FUNCTION_BLOCK AxisControl
VAR
	
	// Axis Reference
	_Axis					: ARRAY [1.._NumberOfAxes] OF AXIS_REF;		
	
	// Internal Variables
	_i						: UINT := 0;
	_InputToggle			: BOOL := FALSE;
	_LocalState				: UINT := 0;
	_InternalCounter		: UDINT := 0;
	_InternalCounterMax		: UDINT := 1000;
	_ErrorIDPrevious		: ARRAY [1.._NumberOfAxes] OF UDINT;
	_ErrorCount				: ARRAY [1.._NumberOfAxes] OF UINT;
	_BusyMoving				: ARRAY [1.._NumberOfAxes] OF BOOL;
	_BusyStopping			: ARRAY [1.._NumberOfAxes] OF BOOL;
	_CommandDone			: BOOL := FALSE;
	_CurrentPosition		: ARRAY [1.._NumberOfAxes] OF LREAL;
	_CurrentPositionModulo	: ARRAY [1.._NumberOfAxes] OF LREAL;
	
	// Internal Functions
	_ErrorCountTrigger		: R_TRIG;
	_DelayTimer				: TON;	
	
	// Axis States (STRUCTURE Declaration)
	_Status					: ARRAY [1.._NumberOfAxes] OF AxisStatus;
	
	// Motion Functions Blocks
	_Enable					: ARRAY [1.._NumberOfAxes] OF MC_Power;
	_Reset					: ARRAY [1.._NumberOfAxes] OF MC_Reset;
	_ReadStatus				: ARRAY [1.._NumberOfAxes] OF MC_ReadStatus;
	_WriteParameter			: MC_WriteParameter;	
	_MoveAbs1				: MC_MoveAbsolute;
	_MoveAbs2				: MC_MoveAbsolute;
	_MoveRel1				: MC_MoveRelative;
	_MoveRel2				: MC_MoveRelative;
	_MoveVel1				: MC_MoveVelocity;
	_MoveVel2				: MC_MoveVelocity;
	_StopWeak				: MC_Halt;
	_StopStrong				: MC_Stop;
		
END_VAR
VAR CONSTANT
	
	_NumberOfAxes			: UINT := 3;

END_VAR

METHOD AutoErrorCheckAndReset : BOOL
VAR_INPUT
	AxisID			: UINT;	
END_VAR

// Automatically check for errors on the NC axis, then reset them
// Use with caution, this could cause damage to a physical system if implemented without care

_ReadStatus[AxisID](Axis := _Axis[AxisID]);
_Reset[AxisID](Axis := _Axis[AxisID]);
_ErrorCountTrigger(CLK := _Status[AxisID]._Error);

IF _ErrorCountTrigger.Q THEN
	_ErrorCount[AxisID] := _ErrorCount[AxisID] + 1;
END_IF

IF _Status[AxisID]._Error THEN
	_LocalState := 0;
	_Reset[AxisID].Execute := TRUE;
	IF _Reset[AxisID].Done THEN
		_Reset[AxisID].Execute := FALSE;
		AutoErrorCheckAndReset := TRUE;
	END_IF
END_IF
END_METHOD

PROPERTY AxisStatus : ARRAY [1.._NumberOfAxes] OF AxisStatus
GET
AxisStatus := _Status;
END_GET
SET
END_SET
END_PROPERTY

METHOD CheckForErrors : BOOL
VAR_INPUT	
	AxisID			: UINT;
END_VAR

// Check for errors on the NC axis

_ReadStatus[AxisID](Axis := _Axis[AxisID]);
_ErrorCountTrigger(CLK := _Status[AxisID]._Error);

IF _ErrorCountTrigger.Q THEN
	_ErrorCount[AxisID] := _ErrorCount[AxisID] + 1;
END_IF

IF _Status[AxisID]._Error THEN
	_LocalState := 0;
	CheckForErrors := TRUE;
END_IF
END_METHOD

PROPERTY CurrentPosition : ARRAY [1.._NumberOfAxes] OF LREAL
GET
CurrentPosition := _CurrentPosition;
END_GET
SET
END_SET
END_PROPERTY

PROPERTY CurrentPositionModulo : ARRAY [1.._NumberOfAxes] OF LREAL
GET
CurrentPositionModulo := _CurrentPositionModulo;
END_GET
SET
END_SET
END_PROPERTY

METHOD CyclicUpdate : BOOL
VAR_INPUT
END_VAR

// Update method needs to be called cyclically

_InputToggle := NOT(_InputToggle);

FOR _i := 1 TO _NumberOfAxes DO
	
	_Enable[_i]		(Axis := _Axis[_i]);
	_Reset[_i]		(Axis := _Axis[_i]);
	
	_ReadStatus[_i]
	(
		Axis 					:= _Axis[_i],
		Enable 					:= TRUE,
		Error 					=> _Status[_i]._Error,
		ErrorID 				=> _Status[_i]._ErrorID,
		ErrorStop 				=> _Status[_i]._ErrorStop,
		Disabled 				=> _Status[_i]._Disabled,
		Stopping 				=> _Status[_i]._Stopping,
		StandStill 				=> _Status[_i]._StandStill,
		DiscreteMotion 			=> _Status[_i]._DiscreteMotion,
		ContinuousMotion 		=> _Status[_i]._ContinuousMotion,
		SynchronizedMotion	 	=> _Status[_i]._SynchronizedMotion,
		Homing 					=> _Status[_i]._Homing,
		ConstantVelocity		=> _Status[_i]._ConstantVelocity,
		Accelerating 			=> _Status[_i]._Accelerating,
		Decelerating 			=> _Status[_i]._Decelerating,
		Status 					=> _Status[_i]._Status
	);
	
	_BusyMoving[_i] :=
	(
		_ReadStatus[_i].DiscreteMotion OR
		_ReadStatus[_i].ConstantVelocity OR
		_ReadStatus[_i].SynchronizedMotion
	);
	
	_BusyStopping[_i] :=
	(
		_ReadStatus[_i].Stopping
	);
	
	IF _Status[_i]._ErrorID <> 0 THEN
		_ErrorIDPrevious[_i] := _Status[_i]._ErrorID;
	END_IF
			
	_CurrentPosition[_i] := _Axis[_i].NcToPlc.ActPos;
	_CurrentPositionModulo[_i] := _Axis[_i].NcToPlc.ModuloActPos;
	
END_FOR

CyclicUpdate := TRUE;
END_METHOD

PROPERTY ErrorCount : ARRAY [1.._NumberOfAxes] OF UINT
GET
ErrorCount := _ErrorCount;
END_GET
SET
END_SET
END_PROPERTY

METHOD Halt : BOOL
VAR_INPUT
	AxisID			: UINT;
END_VAR

// Halts the axis, NOT locking the axis from further commands during its process

_StopWeak(Axis := _Axis[AxisID]);

_StopWeak.Execute			:= TRUE;

IF _StopWeak.Done THEN
	_StopWeak.Execute := FALSE;
	Halt := TRUE;
END_IF

IF _StopWeak.Error THEN
	_StopWeak.Execute := FALSE;
END_IF
END_METHOD

METHOD MoveAtVelocity : BOOL
VAR_INPUT
	AxisID			: UINT;
	Velocity		: LREAL;
	Direction		: MC_Direction;
END_VAR

// Move at a given speed in a defined direction until a stop command is activated

_MoveVel1(Axis := _Axis[AxisID]);

_MoveVel1.Velocity 			:= Velocity;
_MoveVel1.Direction			:= Direction;
_MoveVel1.Execute			:= TRUE;

IF _BusyMoving[AxisID] THEN
	_MoveVel1.Execute := FALSE;
	MoveAtVelocity := TRUE;
END_IF

IF _MoveVel1.Error THEN
	_MoveVel1.Execute := FALSE;
	MoveAtVelocity := FALSE;
END_IF
END_METHOD

METHOD MoveToPosition : BOOL
VAR_INPUT
	AxisID			: UINT;
	Position		: LREAL;
	Velocity		: LREAL;
END_VAR

// Move to a specific location at a given speed

_MoveAbs1(Axis := _Axis[AxisID]);

_MoveAbs1.Position			:= Position;
_MoveAbs1.Velocity 			:= Velocity;
_MoveAbs1.Execute			:= TRUE;

IF _MoveAbs1.Done THEN
	_MoveAbs1.Execute := FALSE;
	MoveToPosition := TRUE;
END_IF

IF _MoveAbs1.Error THEN
	_MoveAbs1.Execute := FALSE;
END_IF
END_METHOD

METHOD PowerOff : BOOL
VAR_INPUT
	Override	 	: LREAL;
	AxisID			: UINT;
END_VAR

// Disable the axis

IF Override < 0 THEN
	Override := 0;
ELSIF Override > 100 THEN
	Override := 100;	
END_IF

IF AxisID < 1 THEN
	AxisID := 1;
ELSIF AxisID > _NumberOfAxes THEN
	AxisID := 1;	
END_IF

_Enable[AxisID](Axis := _Axis[AxisID]);

_Enable[AxisID].Enable 				:= FALSE;
_Enable[AxisID].Enable_Negative 	:= FALSE;
_Enable[AxisID].Enable_Positive 	:= FALSE;
_Enable[AxisID].Override 			:= 0;

IF NOT(_Enable[AxisID].Status) THEN
	PowerOff := TRUE;
ELSIF _Enable[AxisID].Error THEN
	PowerOff := FALSE;
	_Enable[AxisID].Enable := FALSE;
END_IF
END_METHOD

METHOD PowerOffAll : BOOL
VAR_INPUT
END_VAR

// Enable all axes

FOR _i := 1 TO _NumberOfAxes BY 1 DO
	_Enable[_i](Axis := _Axis[_i]);
END_FOR

CASE _LocalState OF 
	
	0:
		_LocalState := 1;
	
	1:
		FOR _i := 1 TO _NumberOfAxes BY 1 DO
			_Enable[_i](Axis := _Axis[_i]);
			_Enable[_i].Enable := FALSE;
			_Enable[_i].Enable_Negative := FALSE;
			_Enable[_i].Enable_Positive := FALSE;
			_Enable[_i].Override := 0;
		END_FOR
		_LocalState := 2;
		
	2:
		_CommandDone := TRUE;
		FOR _i := 1 TO _NumberOfAxes BY 1 DO
			IF _Enable[_i].Status THEN
				_CommandDone := FALSE;
				_InternalCounter := _InternalCounter + 1;
			END_IF
		END_FOR
		
		IF _InternalCounter >= _InternalCounterMax THEN
			_InternalCounter := 0;
			_LocalState := 0;
			PowerOffAll := FALSE;
		END_IF
		
		IF _CommandDone THEN
			_InternalCounter := 0;
			_LocalState := 3;
		END_IF
		
	3:
		_LocalState := 0;
		PowerOffAll := TRUE;

END_CASE
END_METHOD

METHOD PowerOn : BOOL
VAR_INPUT
	Override	 	: LREAL;
	AxisID			: UINT;
END_VAR

// Enable the axis

IF Override < 0 THEN
	Override := 0;
ELSIF Override > 100 THEN
	Override := 100;	
END_IF

IF AxisID < 1 THEN
	AxisID := 1;
ELSIF AxisID > _NumberOfAxes THEN
	AxisID := 1;	
END_IF

_Enable[AxisID](Axis := _Axis[AxisID]);

_Enable[AxisID].Enable 				:= TRUE;
_Enable[AxisID].Enable_Negative 	:= TRUE;
_Enable[AxisID].Enable_Positive 	:= TRUE;
_Enable[AxisID].Override 			:= 100;

IF _Enable[AxisID].Status THEN
	PowerOn := TRUE;
ELSIF _Enable[AxisID].Error THEN
	PowerOn := FALSE;
	_Enable[AxisID].Enable := FALSE;
END_IF
END_METHOD

METHOD PowerOnAll : BOOL
VAR_INPUT
	Override		: LREAL;
END_VAR

// Enable all axes

IF Override < 0 THEN
	Override := 0;
ELSIF Override > 100 THEN
	Override := 100;	
END_IF

FOR _i := 1 TO _NumberOfAxes BY 1 DO
	_Enable[_i](Axis := _Axis[_i]);
END_FOR

CASE _LocalState OF 
	
	0:
		_LocalState := 1;
	
	1:
		FOR _i := 1 TO _NumberOfAxes BY 1 DO
			_Enable[_i](Axis := _Axis[_i]);
			_Enable[_i].Enable := TRUE;
			_Enable[_i].Enable_Negative := TRUE;
			_Enable[_i].Enable_Positive := TRUE;
			_Enable[_i].Override := Override;
		END_FOR
		_LocalState := 2;
		
	2:
		_CommandDone := TRUE;
		FOR _i := 1 TO _NumberOfAxes BY 1 DO
			IF NOT(_Enable[_i].Status) THEN
				_CommandDone := FALSE;
				_InternalCounter := _InternalCounter + 1;
			END_IF
		END_FOR
		
		IF _InternalCounter >= _InternalCounterMax THEN
			_InternalCounter := 0;
			_LocalState := 0;
			PowerOnAll := FALSE;
		END_IF
		
		IF _CommandDone THEN
			_InternalCounter := 0;
			_LocalState := 3;
		END_IF
		
	3:
		_LocalState := 0;
		PowerOnAll := TRUE;

END_CASE
END_METHOD

METHOD Reset : BOOL
VAR_INPUT
	AxisID			: UINT;
END_VAR

// Reset errors on the NC axis

IF AxisID < 1 THEN
	AxisID := 1;
ELSIF AxisID > _NumberOfAxes THEN
	AxisID := 1;	
END_IF

_Reset[AxisID](Axis := _Axis[AxisID]);

_Reset[AxisID].Execute 			:= TRUE;

IF _Reset[AxisID].Done THEN
	_Reset[AxisID].Execute := FALSE;
	Reset := TRUE;
END_IF
END_METHOD

METHOD ReversingSequence : BOOL
VAR_INPUT
	AxisID			: UINT;
	Position1				: LREAL;
	Position2				: LREAL;
	Velocity				: LREAL;
	DelayBetweenMoves		: TIME;
END_VAR

// Move to Position1, then to Position2, at a set speed with a delay between the movements

_MoveAbs1(Axis := _Axis[AxisID]);
_MoveAbs2(Axis := _Axis[AxisID]);
_DelayTimer(PT := DelayBetweenMoves);

_MoveAbs1.Position			:= Position1;
_MoveAbs1.Velocity 			:= Velocity;

_MoveAbs2.Position			:= Position2;
_MoveAbs2.Velocity 			:= Velocity;

CASE _LocalState OF
	
	0:
		_MoveAbs1.Execute := TRUE;
		IF _MoveAbs1.Done THEN
			_MoveAbs1.Execute := FALSE;
			_LocalState := 1;			
		END_IF
		
	1:
		_DelayTimer.IN := TRUE;
		IF _DelayTimer.Q THEN
			_DelayTimer.IN := FALSE;
			_LocalState := 2;
		END_IF
		
	2:
		_MoveAbs2.Execute := TRUE;
		IF _MoveAbs2.Done THEN
			_MoveAbs2.Execute := FALSE;
			_LocalState := 3;			
		END_IF
		
	3:
		_DelayTimer.IN := TRUE;
		IF _DelayTimer.Q THEN
			_DelayTimer.IN := FALSE;
			_LocalState := 4;
		END_IF
		
	4:
		_LocalState := 0;
		ReversingSequence := TRUE;

END_CASE

IF _MoveAbs1.Error OR _MoveAbs2.Error THEN
	_MoveAbs1.Execute := FALSE;
	_MoveAbs2.Execute := FALSE;
END_IF
END_METHOD

METHOD Stop : BOOL
VAR_INPUT
	AxisID			: UINT;
END_VAR

// Halts the axis, locking the axis from further commands during its process

_StopStrong(Axis := _Axis[AxisID]);

_StopStrong.Execute			:= TRUE;

IF _StopStrong.Done THEN
	_StopStrong.Execute := FALSE;
	Stop := TRUE;
END_IF

IF _StopStrong.Error THEN
	_StopStrong.Execute := FALSE;
END_IF
END_METHOD

METHOD WriteToParameter : BOOL
VAR_INPUT
	AxisID			: UINT;	
	Parameter		: MC_AxisParameter;
	Value			: LREAL;
END_VAR

IF AxisID < 1 THEN
	AxisID := 1;
ELSIF AxisID > _NumberOfAxes THEN
	AxisID := 1;	
END_IF

_WriteParameter(Axis := _Axis[AxisID]);

_WriteParameter.ParameterNumber := Parameter;
_WriteParameter.Value := Value;
_WriteParameter.Execute := TRUE;


IF _WriteParameter.Done THEN
	WriteToParameter := TRUE;
	_WriteParameter.Execute := FALSE;
ELSIF _WriteParameter.Error THEN
	WriteToParameter := FALSE;
	_WriteParameter.Execute := FALSE;
END_IF
END_METHOD

END_FUNCTION_BLOCK

(* stored: Version 1.1.0.1, ProductVersion 3.1.4024.12
   POU AxisControl: Id {0762ff6d-63f2-4251-b923-cf396e8d588b}, SpecialFunc None
   Folder Methods: Id {84cb375e-4310-4c8e-b285-59f1b782ddd6}
   Folder All Axes: Id {e7566577-33ba-4fd4-a911-8164896a8c57}
   Folder Power and Monitoring: Id {72185a63-bd61-464d-9ba5-7925e55fb430}
   Folder Single Axis: Id {6793107f-f025-4746-9720-75111f89ad08}
   Folder Movements: Id {6fc24c7c-89c4-4f59-a059-62fbfee907d6}
   Folder Brake: Id {531eff0b-604f-4c37-ace9-2958971ea826}
   Folder Position: Id {8d7c9616-e265-4389-960e-a02f0ff11726}
   Folder Velocity: Id {bd356ce1-0682-451a-8f8f-f2d75631abf0}
   Folder Power and Monitoring: Id {dada0367-7150-48df-9b09-3250334c5191}
   Folder Properties: Id {391590a4-d10f-4e23-95ce-50d1b79d7756}
   Method AutoErrorCheckAndReset: Id {c4558794-dce0-4723-8ae5-ffe53ab7450c}
   Property AxisStatus: Id {743488a2-70c8-43fc-bb97-edf6af21b812}
   Get Get: Id {c75450e0-e73c-4f6d-987f-cb307a38ed66}
   Set Set: Id {10fca8b1-77ef-4bc2-af4d-2836594ff324}
   Method CheckForErrors: Id {1156e6bc-6693-4a8a-8e9b-2040f7a304f7}
   Property CurrentPosition: Id {0d1e2e23-bb07-4506-9aeb-9d8a3f1ee275}
   Get Get: Id {da39f4b5-331e-4c86-bc7c-08dd1f53b62a}
   Set Set: Id {2634205a-da86-4017-b85e-f528dc45565c}
   Property CurrentPositionModulo: Id {e8141d9f-c0d1-4e38-8d71-2c39cd70b6d8}
   Get Get: Id {691176b4-512c-462b-aa59-d8430d3ceba7}
   Set Set: Id {d888dd7e-e7e5-474c-9371-00d8cdc883c5}
   Method CyclicUpdate: Id {176bec90-816f-4a05-8962-1238a59c2f75}
   Property ErrorCount: Id {2a69a2b3-4084-45d9-8c58-9ec4131dbcea}
   Get Get: Id {df5fca3a-d559-4692-b26f-04bdffd38858}
   Set Set: Id {74b040fc-cc77-439a-a040-356ee4860fad}
   Method Halt: Id {12ca4ce0-9928-46fe-8da6-258c70e9b8b4}
   Method MoveAtVelocity: Id {031bd219-54b3-423c-a59d-8808208dd282}
   Method MoveToPosition: Id {6f3dc5db-e33f-4ac2-89b3-444ea6b1636a}
   Method PowerOff: Id {931cb592-80ae-4fd4-9bc7-23c7456ec9bf}
   Method PowerOffAll: Id {9b0e604b-5d41-49b9-90f5-0c685b4b557c}
   Method PowerOn: Id {055fc17f-11ee-4864-95b6-aec8c64cb3a6}
   Method PowerOnAll: Id {093c7e56-b9c1-443e-a0d9-93c4a871420c}
   Method Reset: Id {42cec210-5b3f-4f2e-9099-2c39c8e00b0b}
   Method ReversingSequence: Id {cfe6002d-006b-4fb1-82ee-b56b6ae14ab9}
   Method Stop: Id {e8f89590-5010-45fb-a6e8-5b340988abbd}
   Method WriteToParameter: Id {9cfda403-6e05-479b-94e2-36ef4e728d76} *)
